# EPICS autosave request: trunk/stdApp/Db/femto_DDPCA_300.req
$(P)$(A):Description
$(P)$(A):GainIndex
